Staubli VAL3: getTrajTool.pgx

public program getTrajTool(tool& x_tTool[], num x_nIndex)
begin
  // get the traj tool
  call tcp:getTool(x_tTool,x_nIndex)
end
